FUNCTION CheckBounds : INT
VAR_INPUT
    InValue : INT;
END_VAR
VAR
END_VAR

IF InValue < 15 THEN
    CheckBounds := 15;
ELSIF InValue > 24 THEN
    CheckBounds := 24;
ELSE
    CheckBounds := InValue;
END_IF

END_FUNCTION

(* stored: Version 1.1.0.1, ProductVersion 3.1.4024.15
   POU CheckBounds: Id {16801999-9329-4da5-8fbd-ab12aa941d32}, SpecialFunc None *)
